//<DataManagerDeclarations>
// Function block for data maipulation must extend from TcoData.TcoDataExchange.
FUNCTION_BLOCK TcoDataManagerPlc2 EXTENDS TcoData.TcoDataExchange
VAR
    // This is the structure that contains the actual data we will work with. The `STRUCT` must extend `TcoData.TcoEntity`
    _data : stProcessData_Plc2;
END_VAR
//</DataManagerDeclarations>

//----------------------------------
//<DataManagerSuperCall>
// IMPLEMENTATION BODY OF FUNCTION BLOCK
// IMPORTANT: SUPER CALL HERE IS REQUIRED TO CALL THE DATA MANAGER TASKS!!!
SUPER^();
//</DataManagerSuperCall>
//----------------------------------

PROPERTY Data : REFERENCE TO stProcessData_Plc2
GET
Data REF= _data;
END_GET
END_PROPERTY

END_FUNCTION_BLOCK

(* stored: Version 1.1.0.1, ProductVersion 3.1.4024.12
   POU TcoDataManagerPlc2: Id {7f2c29b4-5945-0f8a-0265-483f7728ce61}, SpecialFunc None
   Property Data: Id {4507aec0-1a86-0024-1ed7-c00ff9cadd07}
   Get Get: Id {13afbc6d-e055-0b4f-0ce3-f97a5f92b723} *)
